(*
SPDX-FileCopyrightText: © 2026 Oleksandr Tiutyk <trofimich@gmail.com>
SPDX-License-Identifier: MIT
License: https://opensource.org/license/mit
*)

(*!
<summary>Dynamic descendants are owned by DynamicMemoryManager until cleanup; static instances remain caller-owned.</summary>
<description>
Clone implementations must return an IException-compatible object; clients borrow registered clones.
</description>
*)

{attribute 'enable_dynamic_creation'}	
{attribute 'no_explicit_call' := 'do not call this function block directly'} 


FUNCTION_BLOCK ABSTRACT Exception EXTENDS Object IMPLEMENTS IException
VAR
	_SourceFullPOUName : STRING(128);
	_SourcePosition : STRING(32);
	_LocalTimestamp : LDATE_AND_TIME;	
	_UtcTimestamp : LDATE_AND_TIME;	
	
	_AutoDisposeRegistrar : AutoDisposeRegistrar(THIS^);
END_VAR

METHOD PROTECTED AppendTimestampDescription
VAR_IN_OUT CONSTANT
	stringBuilder : WideStringBuilder;
END_VAR
VAR_INPUT
	timestampDisplayMode : TIMESTAMP_DISPLAY_MODE := TIMESTAMP_DISPLAY_MODE.HIDDEN;
	localTimestamp : LDATE_AND_TIME;	
	utcTimestamp : LDATE_AND_TIME;	
END_VAR
VAR
	timeStampString : WSTRING(40);
END_VAR
IF timestampDisplayMode = TIMESTAMP_DISPLAY_MODE.HIDDEN THEN
	RETURN;
END_IF

CASE timestampDisplayMode OF
	TIMESTAMP_DISPLAY_MODE.LOCAL:
		timeStampString := TO_WSTRING(localTimestamp);
	
	TIMESTAMP_DISPLAY_MODE.UTC:
		timeStampString := TO_WSTRING(utcTimestamp);
END_CASE

timeStampString := Tc2_Standard.WLEFT(Tc2_Standard.WDELETE(timeStampString, 4, 1), 22);

stringBuilder.AppendString(timeStampString);
IF timestampDisplayMode = TIMESTAMP_DISPLAY_MODE.UTC THEN
	stringBuilder.AppendString("UTC");
END_IF
END_METHOD

(*!
<summary>Resets source and timestamps. Descendants clear their own payload and call this implementation.</summary>
<description>
Does not delete the instance or unregister it from automatic cleanup.
</description>
*)

METHOD Clear
_SourceFullPOUName := '';
_SourcePosition := '';
_LocalTimestamp := LongDateAndTimes.MIN_VALUE;	
_UtcTimestamp := LongDateAndTimes.MIN_VALUE;
END_METHOD

METHOD ABSTRACT Clone : IObject
END_METHOD

{attribute 'monitoring' := 'call'}
PROPERTY ABSTRACT Empty : BOOL
GET
END_GET
END_PROPERTY

METHOD PROTECTED ExtractClassName : STRING
VAR_IN_OUT CONSTANT
	sourcePOUName : STRING;
END_VAR
VAR
	splitter : StringSplittingEnumerator;
END_VAR
splitter := Strings.CreateSplitter(sourcePOUName, '.', 0, TRUE, TRUE);

WHILE splitter.MoveNext() DO		
	ExtractClassName := splitter.CurrentEntry;
	
	RETURN;
END_WHILE
END_METHOD

METHOD PROTECTED ExtractMethodName : STRING
VAR_IN_OUT CONSTANT
	sourcePOUName : STRING;
END_VAR
VAR
	splitter : StringSplittingEnumerator;
END_VAR
splitter := Strings.CreateSplitter(sourcePOUName, '.', 0, TRUE, TRUE);

WHILE splitter.MoveNext() DO
	ExtractMethodName := splitter.CurrentEntry;
END_WHILE
END_METHOD

//!<param name="bInCopyCode">if TRUE, the exit method is called for exiting an instance that is copied afterwards (online change).</param>

METHOD FB_exit : BOOL
VAR_INPUT
	
	bInCopyCode	: BOOL;
END_VAR
Clear();
END_METHOD

METHOD PROTECTED GetFullPOUName : STRING(128)
VAR_IN_OUT CONSTANT
	sourceNamespaceName : STRING;
	sourceClassName : STRING;
	sourcePOUName : STRING;
END_VAR
IF sourceNamespaceName <> Strings.Empty THEN
	Strings.AppendToTarget(GetFullPOUName, sourceNamespaceName);
	Strings.AppendToTarget(GetFullPOUName, '.');	
END_IF

IF sourceClassName <> Strings.Empty THEN
	Strings.AppendToTarget(GetFullPOUName, sourceClassName);
	Strings.AppendToTarget(GetFullPOUName, '.');	
	Strings.AppendToTarget255(GetFullPOUName, ExtractMethodName(sourcePOUName));	
	Strings.AppendToTarget(GetFullPOUName, '()');
ELSE
	Strings.AppendToTarget(GetFullPOUName, sourcePOUName);
END_IF
END_METHOD

METHOD ABSTRACT GetMessage : ERROR_MESSAGE
VAR_INPUT
	showSource : BOOL := FALSE;
	timestampDisplayMode : TIMESTAMP_DISPLAY_MODE := TIMESTAMP_DISPLAY_MODE.HIDDEN;
END_VAR
END_METHOD

METHOD ABSTRACT GetRootException : IException
END_METHOD

METHOD GetSourceDescription : STRING(255)
VAR
	stringBuilder : WideStringBuilder;
	
	result : WSTRING(255);
END_VAR
stringBuilder
	.AppendString255(TO_WSTRING(_SourceFullPOUName))
	.AppendStringIf(Exceptions.SOURCE_POSITION_PREFIX, sourcePosition <> '')
	.AppendString255If(TO_WSTRING(sourcePosition), sourcePosition <> '')
	.AssignToString(result);

GetSourceDescription := TO_STRING(result);
END_METHOD

{attribute 'monitoring' := 'call'}
PROPERTY FINAL LocalTimestamp : LDATE_AND_TIME
GET
LocalTimestamp := _LocalTimestamp;
END_GET
SET // PROTECTED
_LocalTimestamp := LocalTimestamp;
END_SET
END_PROPERTY

{attribute 'monitoring' := 'call'}
PROPERTY FINAL SourceFullPOUName : REFERENCE TO STRING(128)
GET
SourceFullPOUName REF= _SourceFullPOUName;
END_GET
END_PROPERTY

{attribute 'monitoring' := 'call'}
PROPERTY FINAL SourcePosition : REFERENCE TO STRING(32)
GET
SourcePosition REF= _SourcePosition;
END_GET
END_PROPERTY

METHOD ToError
VAR_IN_OUT CONSTANT
	targetError : ERROR;
END_VAR
VAR_INPUT
	severity : ERROR_SEVERITY;	
END_VAR
IF NOT __ISVALIDREF(targetError) THEN
	RETURN;
END_IF

targetError.Fill(
	severity,
	GetSourceDescription(),
	GetSourceDescription(),
	GetMessage(),
	GetMessage(),
	LocalTimestamp,
	UtcTimestamp
);
END_METHOD

{attribute 'monitoring' := 'call'}
PROPERTY FINAL UtcTimestamp : LDATE_AND_TIME
GET
UtcTimestamp := _UtcTimestamp;
END_GET
SET // PROTECTED
_UtcTimestamp := UtcTimestamp;
END_SET
END_PROPERTY

END_FUNCTION_BLOCK

(* stored: Version 1.1.0.1
   POU Exception: Id {54495eb3-7b3a-47b9-85cb-0393f41c20d3}, SpecialFunc None
   Folder Service members: Id {a47a20ca-4953-4e09-8f4d-fc2e8d3ac96e}
   Method AppendTimestampDescription: Id {a316d3b4-0094-41d5-a4cb-9fba6e2a6883}
   Method Clear: Id {44a047f7-46bd-418c-989f-4458402150ba}
   Method Clone: Id {ff7ec3e0-b6aa-4a29-8b78-e576a86138cb}
   Property Empty: Id {bd97cee3-a16c-4148-a36f-41860b6b4283}
   Get Get: Id {32775313-ab40-46b6-a69f-434f332e1416}
   Method ExtractClassName: Id {2741f852-3263-48be-9dbc-ba747f8558d6}
   Method ExtractMethodName: Id {be44e9a6-255a-48b7-a062-fbf15488833a}
   Method FB_exit: Id {11857425-e8b4-42f5-9cda-87a6242433d1}
   Method GetFullPOUName: Id {55af960f-b27f-4389-9e6d-9c37bf31a838}
   Method GetMessage: Id {6f101456-9a5d-4c21-8b11-8b9151d71824}
   Method GetRootException: Id {14eed042-28c1-47eb-a619-b182b2b0181c}
   Method GetSourceDescription: Id {d08299fd-3dd9-413a-badd-9a2833bcb01e}
   Property LocalTimestamp: Id {4c2d5866-231e-4105-a6bb-6c19851f1e45}
   Get Get: Id {4cb9fd2f-3b41-4625-9c08-af3725cdee6c}
   Set Set: Id {45619644-007a-4d10-a49a-4bb8ab2228ac}
   Property SourceFullPOUName: Id {ce5ba086-21af-4254-a988-84dec5648bcb}
   Get Get: Id {8170787e-91f8-4271-bfce-a70e9b6f9137}
   Property SourcePosition: Id {92080a7c-c630-4b10-82a8-4b95a8267619}
   Get Get: Id {da2e3d95-43f0-4ba4-a676-8010643e418a}
   Method ToError: Id {8d25c83e-d9af-49a8-90c4-2ced5ac3b9ee}
   Property UtcTimestamp: Id {6ae20a8f-f2b2-4c7c-96e2-30787aae9908}
   Get Get: Id {68e22629-e573-41bd-b400-d1cb3c398e1f}
   Set Set: Id {b2d25d91-e13d-48d8-a20e-cde8a5d29fe4} *)
